// Digital sensor
FUNCTION_BLOCK FB_Sensor
VAR_INPUT
	bSignal: BOOL;                 // Signal from the sensor
	eSignalType: eSensorType;      // Type of the sensor: NO, NC
END_VAR
VAR_OUTPUT
END_VAR
VAR
END_VAR

// Sensor is detecting the object 
PROPERTY isFree : Bool
GET
CASE eSignalType OF                          // Set the sensor is occupied state accroding to the type 
	eSensorType.NO: 
		isFree := NOT bSignal;
	eSensorType.NC:
		isFree := bSignal;
END_CASE
END_GET
END_PROPERTY

// Sensor is not detecting any objects
PROPERTY isOccupied : Bool
GET
CASE eSignalType OF             // Set the sensor is free state accroding to the type 
	eSensorType.NO:
		isOccupied := bSignal;
	eSensorType.NC:
		isOccupied := NOT bSignal;
END_CASE
END_GET
END_PROPERTY

END_FUNCTION_BLOCK

(* stored: Version 1.1.0.1, ProductVersion 3.1.4024.12
   POU FB_Sensor: Id {692811f0-6506-42e2-94ec-026318027f18}, SpecialFunc None
   Property isFree: Id {aed67602-89bc-4e39-b1f7-32748128792c}
   Get Get: Id {13c78d76-6384-433d-bdfa-94ca5f356fc5}
   Property isOccupied: Id {a8024755-c2f1-4e43-8391-e21a72b9bd04}
   Get Get: Id {04f7ea43-981d-42da-ab71-e1d789fb8eb7} *)
